// modulo (shortest way)/absolute movements
// -- - + ++
// move / pos / velo
// stop / reset
// 
TYPE ST_AxisControlLS :
STRUCT
	bLimitSwitchStateMin						: BOOL;
	bLimitSwitchStateMax						: BOOL;
	bWriteLS									: BOOL;
	bReadLS										: BOOL;
	fLimitSwitchPositionMax						: LREAL;
	fLimitSwitchPositionMin						: LREAL;
END_STRUCT
END_TYPE

(* stored: Version 1.2.0.0, ProductVersion 3.1.4026.13, FileIdentifier 3ed7e6e4a20d34d03043445aa9b3e292abf2e5a4, FileSignature 35c45d7110344b057adca989f394453b5f2b16f8fbda7819f323bd50b99d4a168ba4a8bbfa801ef3afac49fb77d2d6b9a599345e827ef5e45e7a850e0b4f63c98f9795faadf021bf068f01a8efa9448f4f996ce8a496a7fc0c7b3de1f15a95520941e17e1e41f52839af4c31f2f6e9f772aed6551bfc087279878326ff17d4c367edcab1e46d350101ebe9a5e373b8ff430aa0db21dd309c0a4925e20570d199674f6e675f2919de6155143f9058fb691ff4fc7bb2ab7a00d693958c9e1edf53ff50ea04de8bca9071d14b7f8febff712ab312b07be64dce8dd0584c3a30255b6d210cee86db61d3730241a8cff730ccccaa8c8308b374c4e4c54679afeaeade
   DUT ST_AxisControlLS: Id {f2667ea1-f2f7-43f4-a6f2-af50eff50a0e} *)
